// SIMATIC S7-200 project (STEP 7-Micro/WIN), CPU 214 REL 01.11

SYMBOL_TABLE USER1
Start            I0.0     // Start button
Stop_Button      I0.1     // Stop button
Machine_Start    M0.0     // Starting the machine
Restart          M0.1     // Restart the process
RF1              I0.2     // Reflex light beam switch to detect object near meatal sensor
Metal_Sensor     I0.3     // Metal detecting sensor
RF2              I0.4     // Reflex light beam switch to detect object near color sensor
Color_Sensor     I0.5     // Color detecting sensor
S1               I0.6     // Feeding actuator limit
S2               I0.7     // Sorting ejector actuator limit
S3               I1.0     // Other bottle ejectro actuator limit
RF3              I1.1     // Reflex light beam switch to detect object near sorted object ejector
RF4              I1.2     // Reflex light beam switch to detect object near other object ejector
Ejection_Done    M0.2     // Ejection completed
Object           M0.3     // Object introduction bit
Metal_Detecting  M0.4     // Metal detection kick off
Metal_Object     M0.5     // Metal object represent bit
Non_Metal_Object M0.6     // Non metal object represent bit
Metal_Detecting_Done M0.7     // Metal detecting completed
Metal_Sorted     M1.1     // Metal sorting completion represent bit
Color_Detecting  M1.2     // Color detection kick off
Orange_Object    M1.3     // Orange object represent bit
Non_Orange_Object M1.4     // Non orange represent bit
Color_Detecting_Done M1.5     // Color detection completed
Color_Sorted     M1.6     // Color sorting completion represet bit
Sorting_Ejector_Start M1.7     // Sorted bottle ejection kick off
Cycle_Completed  M2.0     // Cycle completion represent bit
Other_Bottle_Ejector_St M2.1     // Other bottle ejection kick off
Motor            Q0.0     // Motor
P1               Q0.1     // Feeding actator forward solenoid
P2               Q0.2     // Sorting ejector actator forward solenoid
P3               Q0.3     // Other bottle ejector actator forward solenoid
END_SYMBOL_TABLE

ORGANIZATION_BLOCK MAIN:OB1
TITLE=PROGRAM COMMENTS
BEGIN
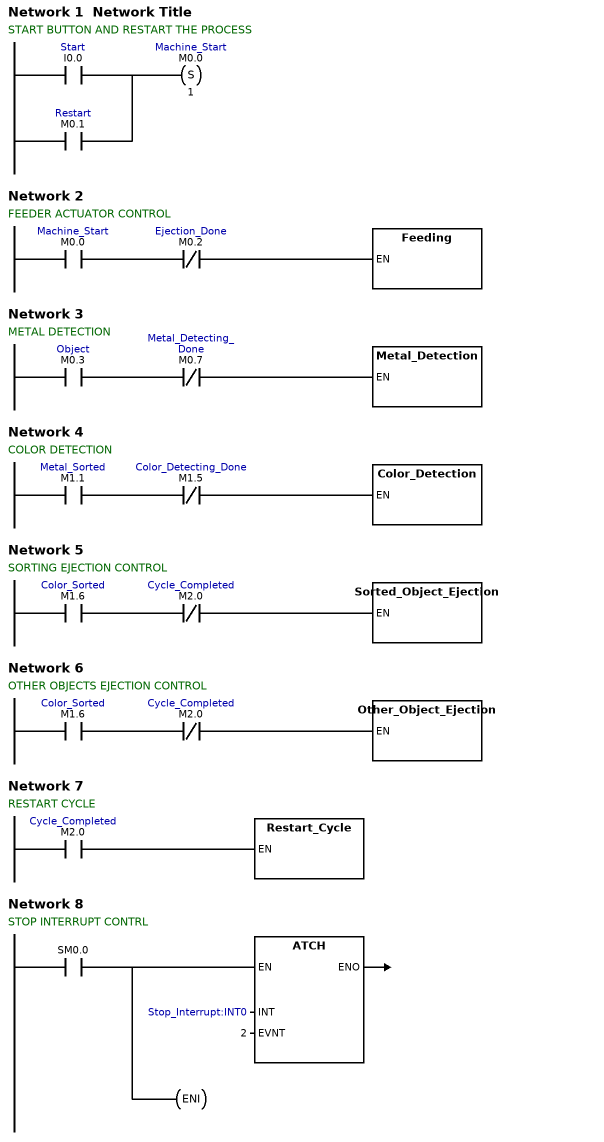
Network 1 // Network Title
// START BUTTON AND RESTART THE PROCESS 
LD     Start:I0.0
O      Restart:M0.1
S      Machine_Start:M0.0, 1
Network 2
// FEEDER ACTUATOR CONTROL
LD     Machine_Start:M0.0
AN     Ejection_Done:M0.2
CALL   Feeding:SBR0
Network 3
// METAL DETECTION 
LD     Object:M0.3
AN     Metal_Detecting_Done:M0.7
CALL   Metal_Detection:SBR1
Network 4
// COLOR DETECTION
LD     Metal_Sorted:M1.1
AN     Color_Detecting_Done:M1.5
CALL   Color_Detection:SBR2
Network 5
// SORTING EJECTION CONTROL
LD     Color_Sorted:M1.6
AN     Cycle_Completed:M2.0
CALL   Sorted_Object_Ejection:SBR3
Network 6
// OTHER OBJECTS EJECTION CONTROL
LD     Color_Sorted:M1.6
AN     Cycle_Completed:M2.0
CALL   Other_Object_Ejection:SBR4
Network 7
// RESTART CYCLE
LD     Cycle_Completed:M2.0
CALL   Restart_Cycle:SBR5
Network 8
// STOP INTERRUPT CONTRL
LD     SM0.0
ATCH   Stop_Interrupt:INT0, 2
ENI
END_ORGANIZATION_BLOCK

SUBROUTINE_BLOCK Feeding:SBR0
TITLE=FEEDING SUBROUTINE
BEGIN
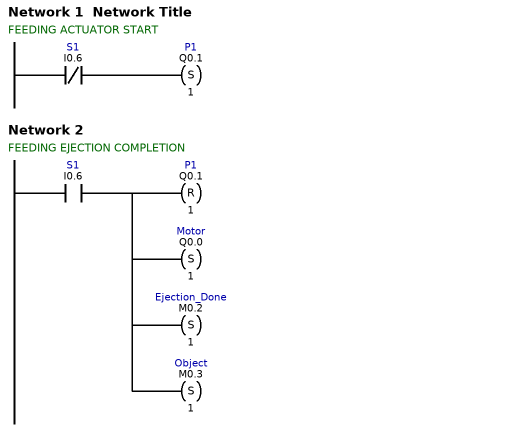
Network 1 // Network Title
// FEEDING ACTUATOR START
LDN    S1:I0.6
S      P1:Q0.1, 1
Network 2
// FEEDING EJECTION COMPLETION
LD     S1:I0.6
R      P1:Q0.1, 1
S      Motor:Q0.0, 1
S      Ejection_Done:M0.2, 1
S      Object:M0.3, 1
END_SUBROUTINE_BLOCK

SUBROUTINE_BLOCK Metal_Detection:SBR1
TITLE=METAL DETECTION
BEGIN
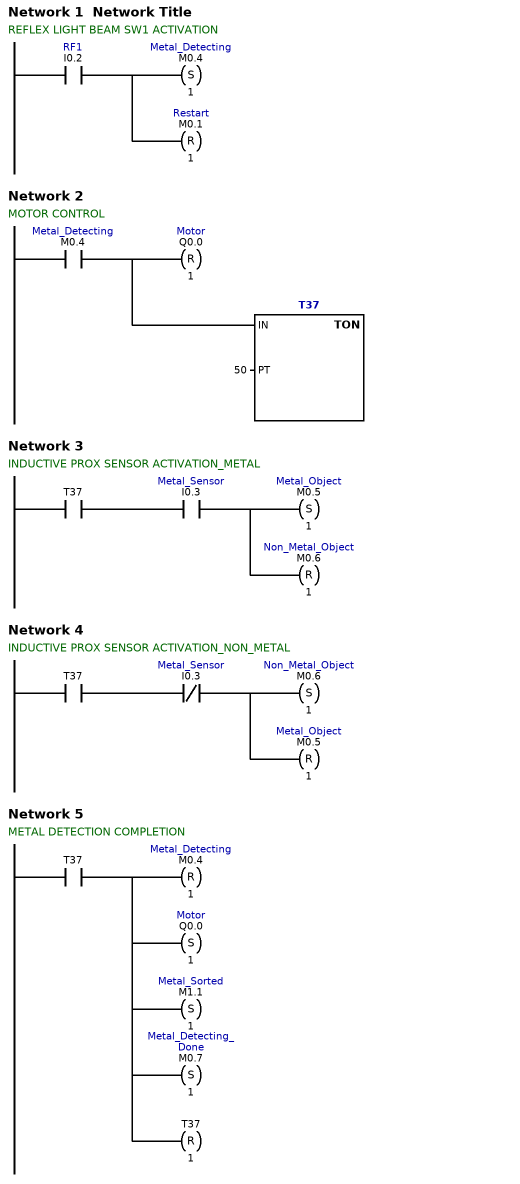
Network 1 // Network Title
// REFLEX LIGHT BEAM SW1 ACTIVATION
LD     RF1:I0.2
S      Metal_Detecting:M0.4, 1
R      Restart:M0.1, 1
Network 2
// MOTOR CONTROL
LD     Metal_Detecting:M0.4
R      Motor:Q0.0, 1
TON    T37, 50
Network 3
// INDUCTIVE PROX SENSOR ACTIVATION_METAL
LD     T37
A      Metal_Sensor:I0.3
S      Metal_Object:M0.5, 1
R      Non_Metal_Object:M0.6, 1
Network 4
// INDUCTIVE PROX SENSOR ACTIVATION_NON_METAL
LD     T37
AN     Metal_Sensor:I0.3
S      Non_Metal_Object:M0.6, 1
R      Metal_Object:M0.5, 1
Network 5
// METAL DETECTION COMPLETION
LD     T37
R      Metal_Detecting:M0.4, 1
S      Motor:Q0.0, 1
S      Metal_Sorted:M1.1, 1
S      Metal_Detecting_Done:M0.7, 1
R      T37, 1
END_SUBROUTINE_BLOCK

SUBROUTINE_BLOCK Color_Detection:SBR2
TITLE=COLOR DETECTION
BEGIN
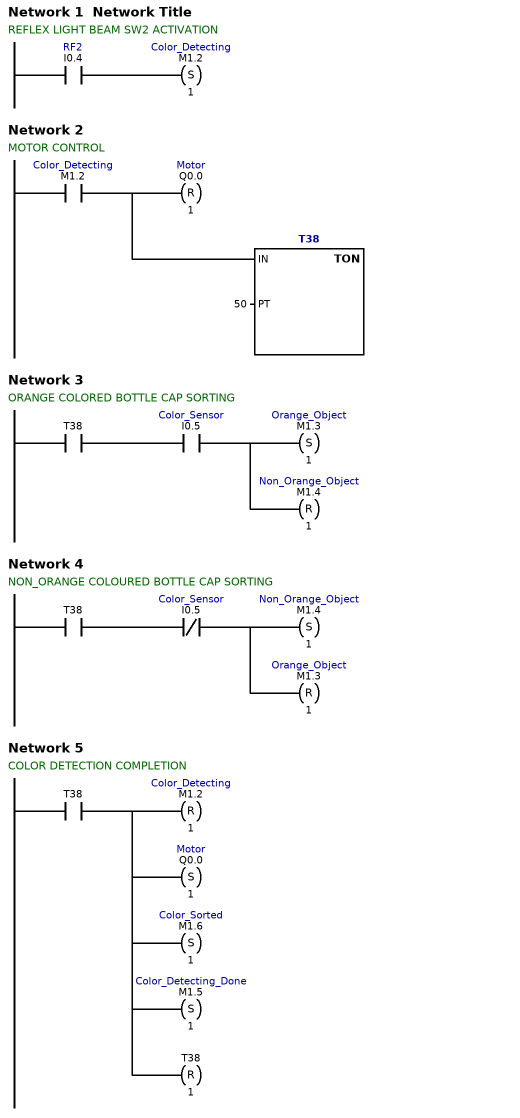
Network 1 // Network Title
// REFLEX LIGHT BEAM SW2 ACTIVATION
LD     RF2:I0.4
S      Color_Detecting:M1.2, 1
Network 2
// MOTOR CONTROL
LD     Color_Detecting:M1.2
R      Motor:Q0.0, 1
TON    T38, 50
Network 3
// ORANGE COLORED BOTTLE CAP SORTING
LD     T38
A      Color_Sensor:I0.5
S      Orange_Object:M1.3, 1
R      Non_Orange_Object:M1.4, 1
Network 4
//  NON_ORANGE COLOURED BOTTLE CAP SORTING
LD     T38
AN     Color_Sensor:I0.5
S      Non_Orange_Object:M1.4, 1
R      Orange_Object:M1.3, 1
Network 5
// COLOR DETECTION COMPLETION
LD     T38
R      Color_Detecting:M1.2, 1
S      Motor:Q0.0, 1
S      Color_Sorted:M1.6, 1
S      Color_Detecting_Done:M1.5, 1
R      T38, 1
END_SUBROUTINE_BLOCK

SUBROUTINE_BLOCK Sorted_Object_Ejection:SBR3
TITLE=SORTED OBJECT EJECTION
BEGIN
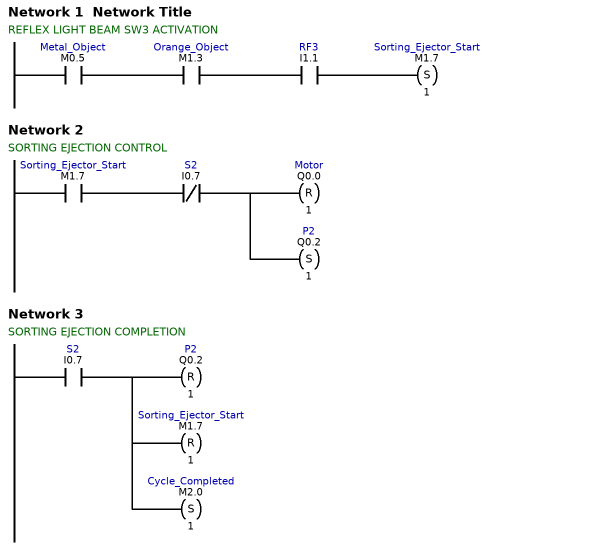
Network 1 // Network Title
// REFLEX LIGHT BEAM SW3 ACTIVATION
LD     Metal_Object:M0.5
A      Orange_Object:M1.3
A      RF3:I1.1
S      Sorting_Ejector_Start:M1.7, 1
Network 2
// SORTING EJECTION CONTROL
LD     Sorting_Ejector_Start:M1.7
AN     S2:I0.7
R      Motor:Q0.0, 1
S      P2:Q0.2, 1
Network 3
// SORTING EJECTION COMPLETION
LD     S2:I0.7
R      P2:Q0.2, 1
R      Sorting_Ejector_Start:M1.7, 1
S      Cycle_Completed:M2.0, 1
END_SUBROUTINE_BLOCK

SUBROUTINE_BLOCK Other_Object_Ejection:SBR4
TITLE=OTHER OBJECT EJECTION
BEGIN
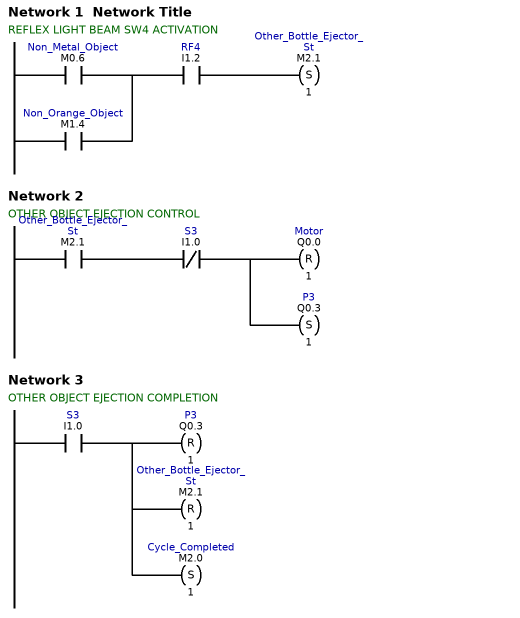
Network 1 // Network Title
// REFLEX LIGHT BEAM SW4 ACTIVATION
LD     Non_Metal_Object:M0.6
O      Non_Orange_Object:M1.4
A      RF4:I1.2
S      Other_Bottle_Ejector_St:M2.1, 1
Network 2
// OTHER OBJECT EJECTION CONTROL
LD     Other_Bottle_Ejector_St:M2.1
AN     S3:I1.0
R      Motor:Q0.0, 1
S      P3:Q0.3, 1
Network 3
// OTHER OBJECT EJECTION COMPLETION
LD     S3:I1.0
R      P3:Q0.3, 1
R      Other_Bottle_Ejector_St:M2.1, 1
S      Cycle_Completed:M2.0, 1
END_SUBROUTINE_BLOCK

SUBROUTINE_BLOCK Restart_Cycle:SBR5
TITLE=RESTART CYCLE
BEGIN
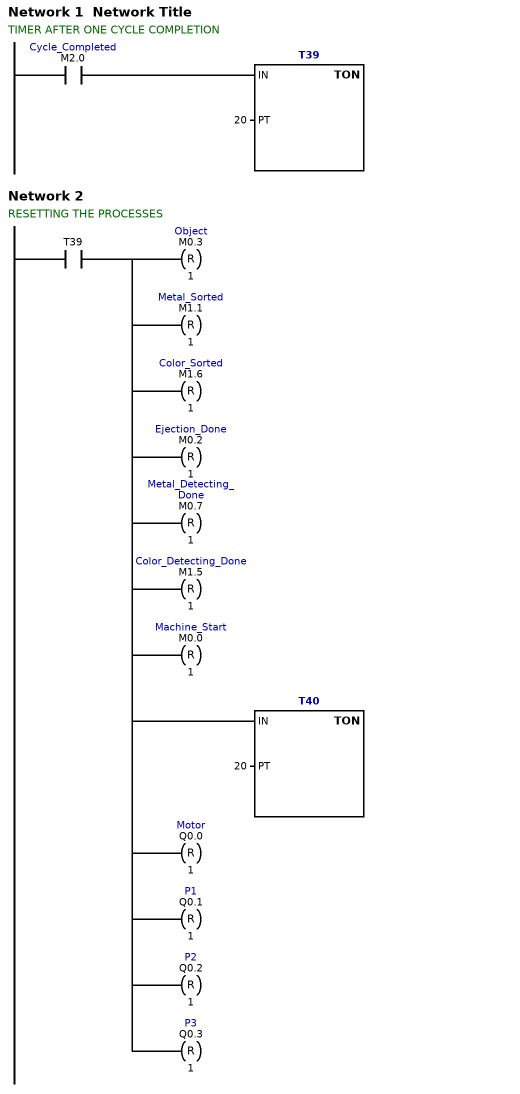
Network 1 // Network Title
// TIMER AFTER ONE CYCLE COMPLETION
LD     Cycle_Completed:M2.0
TON    T39, 20
Network 2
// RESETTING THE PROCESSES
LD     T39
R      Object:M0.3, 1
R      Metal_Sorted:M1.1, 1
R      Color_Sorted:M1.6, 1
R      Ejection_Done:M0.2, 1
R      Metal_Detecting_Done:M0.7, 1
R      Color_Detecting_Done:M1.5, 1
R      Machine_Start:M0.0, 1
TON    T40, 20
R      Motor:Q0.0, 1
R      P1:Q0.1, 1
R      P2:Q0.2, 1
R      P3:Q0.3, 1
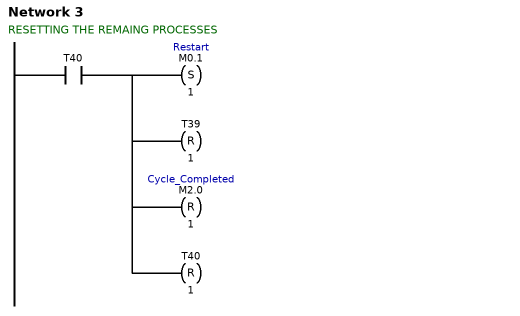
Network 3
// RESETTING THE REMAING PROCESSES
LD     T40
S      Restart:M0.1, 1
R      T39, 1
R      Cycle_Completed:M2.0, 1
R      T40, 1
END_SUBROUTINE_BLOCK

INTERRUPT_BLOCK Stop_Interrupt:INT0
TITLE=STOP INTERRUPT PROCESS
BEGIN
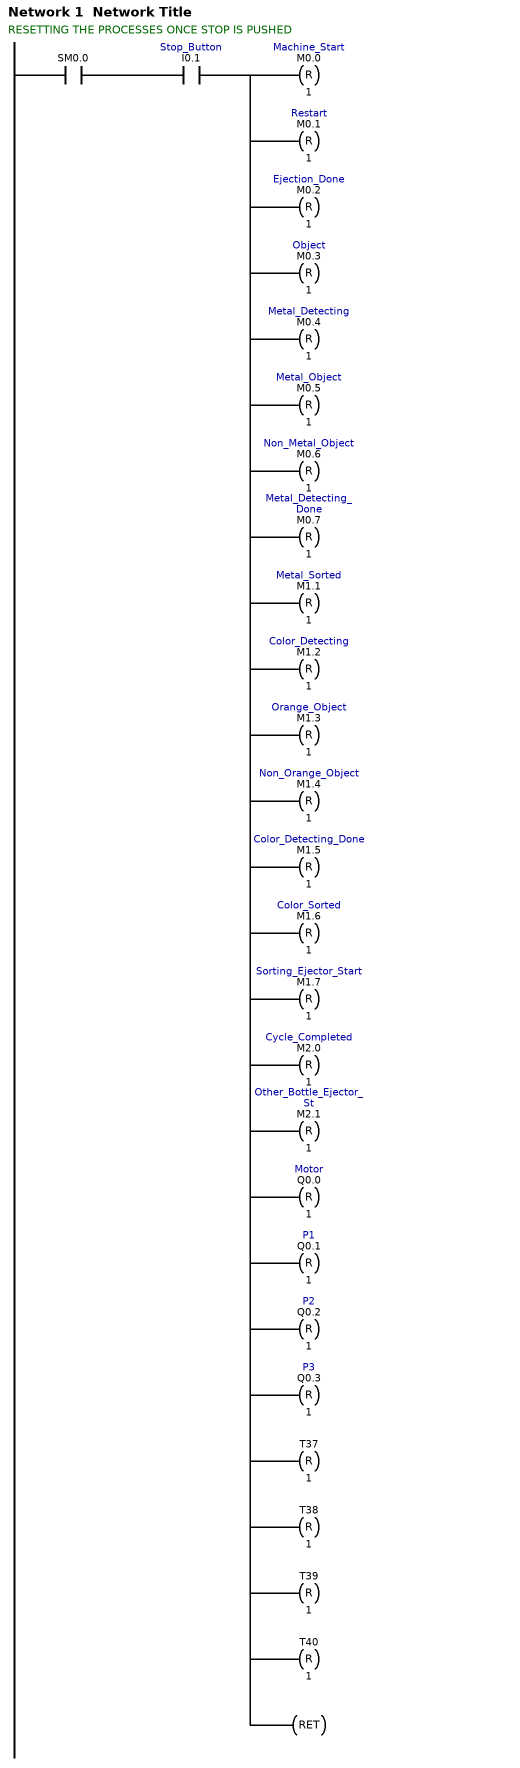
Network 1 // Network Title
// RESETTING THE PROCESSES ONCE STOP IS PUSHED
LD     SM0.0
A      Stop_Button:I0.1
R      Machine_Start:M0.0, 1
R      Restart:M0.1, 1
R      Ejection_Done:M0.2, 1
R      Object:M0.3, 1
R      Metal_Detecting:M0.4, 1
R      Metal_Object:M0.5, 1
R      Non_Metal_Object:M0.6, 1
R      Metal_Detecting_Done:M0.7, 1
R      Metal_Sorted:M1.1, 1
R      Color_Detecting:M1.2, 1
R      Orange_Object:M1.3, 1
R      Non_Orange_Object:M1.4, 1
R      Color_Detecting_Done:M1.5, 1
R      Color_Sorted:M1.6, 1
R      Sorting_Ejector_Start:M1.7, 1
R      Cycle_Completed:M2.0, 1
R      Other_Bottle_Ejector_St:M2.1, 1
R      Motor:Q0.0, 1
R      P1:Q0.1, 1
R      P2:Q0.2, 1
R      P3:Q0.3, 1
R      T37, 1
R      T38, 1
R      T39, 1
R      T40, 1
CRET
Network 2
// RESETTING PROCESSES
Network 3
// RESETTING TIMERS AND REMAING PROCESSES
END_INTERRUPT_BLOCK
